Universal Robots URScript: LensSpacer.script

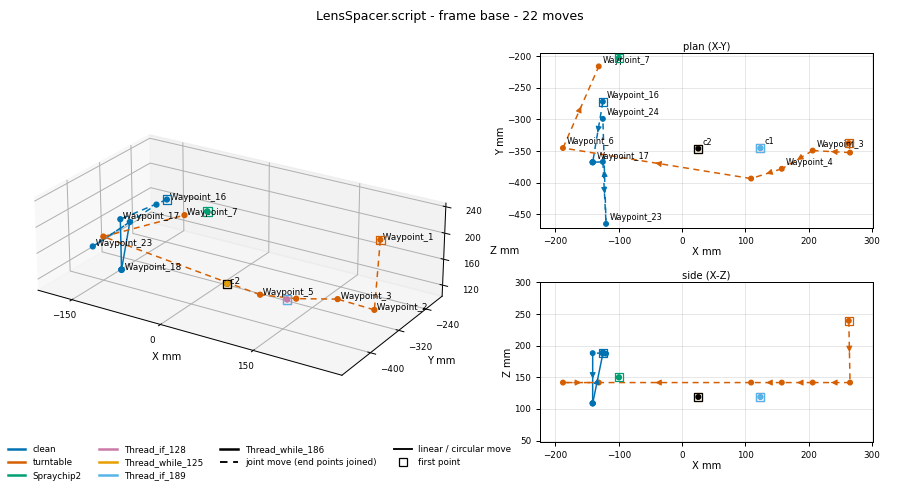
[picture p0: tool path of LensSpacer.script in frame base, 22 of 66 moves have a stored position in this frame; points joined in program order, loops and branches not executed]
def LensSpacer():
  global _hidden_verificationVariable=0
  step_count_fb48d3ff_0c9f_4d99_a765_ea41926c28d5 = 0.0
  thread Step_Counter_Thread_a9617a2c_6c0b_4ca4_aaba_c79477845290():
    while (True):
      step_count_fb48d3ff_0c9f_4d99_a765_ea41926c28d5 = step_count_fb48d3ff_0c9f_4d99_a765_ea41926c28d5 + 1.0
      sync()
    end
  end
  run Step_Counter_Thread_a9617a2c_6c0b_4ca4_aaba_c79477845290()
  set_standard_analog_input_domain(0, 1)
  set_standard_analog_input_domain(1, 1)
  set_tool_analog_input_domain(0, 1)
  set_tool_analog_input_domain(1, 1)
  set_analog_outputdomain(0, 0)
  set_analog_outputdomain(1, 0)
  set_input_actions_to_default()
  set_tool_communication(False, 115200, 0, 1, 1.5, 3.5)
  set_tool_output_mode(0)
  set_tool_digital_output_mode(0, 1)
  set_tool_digital_output_mode(1, 1)
  set_tool_voltage(0)
  set_safety_mode_transition_hardness(1)
  set_gravity([0.0, 0.0, 9.82])
  set_target_payload(0.530000, [0.009000, -0.039000, 0.092000], [0.000534, 0.000534, 0.000534, 0.000000, 0.000000, 0.000000])
  set_tcp(p[0.0,0.0,0.11,0.0,0.0,0.0])
  global Al_plate=p[0.12405209206180495,-0.2666666051843552,0.020008101224669964,-9.276623980477388E-5,1.8107917580596192E-5,3.1233857134705927]
  global Frame2x2=p[0.18266245434305164,-0.34273121659514855,0.026002571110600767,-2.225423529876215E-4,3.0110667546023537E-4,3.1233976058306383]
  global Plane_1=p[0.0,0.0,0.0,0.0,0.0,0.0]
  global URlogoTutorial=p[-0.08178353973148575,-0.3363174165299142,0.04788621506469384,-3.9746155723688456E-5,-3.4682148779121894E-5,-1.5668291789091222]
  global carousel=p[0.13865255139760183,-0.25132593351268107,0.051531504137083003,-4.453572132438073E-5,-1.3071222590669835E-4,-3.1349676625391965]
  global carouselrod=p[0.2020731702281844,-0.34951442511341274,0.1947611446273096,3.139766958234101,-0.10689428010274801,-1.1796370330365635E-5]
  global paper=p[-0.09670794781244417,-0.3283412964648025,0.027665994240809913,-3.2057893450593004E-5,2.867088716161181E-5,-1.6085327915291054]
  global rod=p[0.13368013097420872,-0.41123185103490206,0.09926814901395645,2.2214229924093103,-2.2214158162465862,-2.9165882738638143E-5]
  global timer_1=0
  global c1_p=p[.123835058239, -.345418431995, .118986505182, -3.106795474555, -.465619356567, .000150367177]
  global c1_q=[-0.8607562224017542, -1.7996555767455042, -1.6686586141586304, -1.243450478916504, 1.5722103118896484, 3.55291748046875]
  global c2_p=p[.025685349615, -.346070581208, .119008047533, -3.141142372007, .028389149609, .002727345742]
  global c2_q=[-1.1080010573016565, -1.7158266506590785, -1.7707760334014893, -1.2261001926711579, 1.5707616806030273, 3.621312379837036]
  global Waypoint_16_p=p[-.125097928533, -.271984222044, .188211676824, -3.139810722578, .105446315311, .000070958927]
  global Waypoint_16_q=[-1.5480602423297327, -1.4491210740855713, -1.7099264860153198, -1.552596167927124, 1.5715936422348022, 3.23006010055542]
  global Waypoint_17_p=p[-.141183217597, -.367684006591, .188213447751, 3.139821760490, -.105397104768, -.000067867997]
  global Waypoint_17_q=[-1.597567383443014, -1.8740092716612757, -1.241610050201416, -1.5960084400572718, 1.5719740390777588, 3.1803600788116455]
  global Waypoint_18_p=p[-.141178244459, -.367687282910, .108904454765, 3.139816402425, -.105408093734, -.000060814483]
  global Waypoint_18_q=[-1.5975983778582972, -1.9245020351805628, -1.550661325454712, -1.2364590925029297, 1.5723340511322021, 3.1807193756103516]
  global Waypoint_19_p=p[-.141189357305, -.367687267469, .108915260822, 3.121780755938, .351957921543, -.000099281586]
  global Waypoint_19_q=[-1.5976179281817835, -1.9244748554625453, -1.550661325454712, -1.2364507478526612, 1.572314977645874, 2.889045000076294]
  global Waypoint_20_p=p[-.141176698746, -.367682773595, .108907204798, -3.111042719163, .436975672702, .000063164110]
  global Waypoint_20_q=[-1.5975945631610315, -1.9244939289488734, -1.5506495237350464, -1.2365017098239441, 1.5723340511322021, 3.3926987648010254]
  global Waypoint_21_p=p[-.141174078526, -.367696805030, .108909057026, 3.139786221315, -.105395786134, -.000060564502]
  global Waypoint_21_q=[-1.597586456929342, -1.9245058498778285, -1.5506460666656494, -1.2364399594119568, 1.5723340511322021, 3.1807241439819336]
  global Waypoint_22_p=p[-.125093999497, -.367099400456, .187371407622, 3.139783011421, -.105392168035, -.000053869150]
  global Waypoint_22_q=[-1.5538747946368616, -1.846323629418844, -1.2822730541229248, -1.5829936466612757, 1.5719654560089111, 3.224064588546753]
  global Waypoint_23_p=p[-.120064390322, -.465070651334, .187365924664, 2.700279766902, -.088400420341, .019763045538]
  global Waypoint_23_q=[-1.5412524382220667, -1.9475652180113734, -1.406833291053772, -0.9173591893962403, 1.5603561401367188, 3.2332537174224854]
  global Waypoint_24_p=p[-.125099110421, -.299097154487, .189878767902, 3.139750209928, -.105401717856, -.000111797080]
  global Waypoint_24_q=[-1.550074879323141, -1.5617311683348198, -1.5979981422424316, -1.5518303674510499, 1.5716702938079834, 3.2279696464538574]
  global Waypoint_1_p=p[.263501689877, -.337317763427, .239349489480, 3.139797243720, -.105347053477, -.000037720516]
  global Waypoint_1_q=[-0.5959728399859827, -2.1057659588255824, -0.6533136367797852, -1.9525557957091273, 1.5718059539794922, 4.181682586669922]
  global Waypoint_2_p=p[.265438435610, -.352444474661, .141740907029, 3.139726376264, -.105360108121, -.000022031768]
  global Waypoint_2_q=[-0.6231134573565882, -2.1016999683775843, -1.126999020576477, -1.4828875821879883, 1.5722739696502686, 4.154912948608398]
  global Waypoint_3_p=p[.206441973084, -.349241721273, .141737893294, 3.139734184252, -.105329347268, -.000022485776]
  global Waypoint_3_q=[-0.7073677221881312, -1.9410401783385218, -1.3681066036224365, -1.4024366003325959, 1.5721865892410278, 4.070710182189941]
  global Waypoint_4_p=p[.157616611756, -.378012026932, .141738203587, 3.139764187573, -.105376653239, -.000076760662]
  global Waypoint_4_q=[-0.8494070211993616, -1.9579774341978968, -1.3439116477966309, -1.409730003481247, 1.5722019672393799, 3.928692579269409]
  global Waypoint_5_p=p[.109134761588, -.393436595889, .141742225598, 3.139732501163, -.105376381431, -.000050533951]
  global Waypoint_5_q=[-0.972816292439596, -1.9523960552611292, -1.3519116640090942, -1.4072665137103577, 1.5721949338912964, 3.805286407470703]
  global Waypoint_6_p=p[-.188131250090, -.345166366147, .141750553976, 3.139727051239, -.105353578209, -.000024875816]
  global Waypoint_6_q=[-1.7293437162982386, -1.8864180050291957, -1.4439769983291626, -1.381135032778122, 1.572224736213684, 3.0487747192382812]
  global Waypoint_7_p=p[-.131564048097, -.216205376465, .141741700579, 3.139714533984, -.105382776464, -.000044168049]
  global Waypoint_7_q=[-1.572542969380514, -1.2417927545360108, -2.0833356380462646, -1.3863917154124756, 1.571577787399292, 3.2058310508728027]
  global chipC_p=p[-.099697868296, -.202950013539, .149999031187, 3.139665329235, -.105467028523, -.000070092891]
  global chipC_q=[-1.408487621937887, -1.0837985140136261, -2.130019187927246, -1.497666673069336, 1.571320652961731, 3.369939088821411]
  global timer_1_is_counting=False
  thread Timer_Thread():
    while (True):
      if (timer_1_is_counting):
        timer_1 = timer_1 + get_steptime()
      end
      sync()
    end
  end
  run Timer_Thread()
  def CircleAllangles():
    $ 258 "CircleAllangles" "noBreak"
    $ 259 "p0≔p[c[0]+r,c[1],c[2],c[3],c[4],c[5]-1.5*A]"
    global p0=p[c[0]+r,c[1],c[2],c[3],c[4],c[5]-1.5*A]
    $ 260 "p45≔p[c[0]+0.71*r,c[1]+0.71*r,c[2],c[3]-A/1.1,c[4],c[5]-A/1.1]"
    global p45=p[c[0]+0.71*r,c[1]+0.71*r,c[2],c[3]-A/1.1,c[4],c[5]-A/1.1]
    $ 261 "p90≔p[c[0],c[1]+r,c[2],c[3]-A,c[4],c[5]]"
    global p90=p[c[0],c[1]+r,c[2],c[3]-A,c[4],c[5]]
    $ 262 "p135≔p[c[0]-0.71*r,c[1]+0.71*r,c[2],c[3]-A/1.1,c[4],c[5]+A/1.1]"
    global p135=p[c[0]-0.71*r,c[1]+0.71*r,c[2],c[3]-A/1.1,c[4],c[5]+A/1.1]
    $ 263 "p180≔p[c[0]-r,c[1],c[2],c[3],c[4],c[5]+1.5*A]"
    global p180=p[c[0]-r,c[1],c[2],c[3],c[4],c[5]+1.5*A]
    $ 264 "p225≔p[c[0]-0.71*r,c[1]-0.71*r,c[2],c[3]+A/1.1,c[4],c[5]+A/1.1]"
    global p225=p[c[0]-0.71*r,c[1]-0.71*r,c[2],c[3]+A/1.1,c[4],c[5]+A/1.1]
    $ 265 "p270≔p[c[0],c[1]-r,c[2],c[3]+A,c[4],c[5]]"
    global p270=p[c[0],c[1]-r,c[2],c[3]+A,c[4],c[5]]
    $ 266 "p315≔p[c[0]+0.71*r,c[1]-0.71*r,c[2],c[3]+A/1.1,c[4],c[5]-A/1.1]"
    global p315=p[c[0]+0.71*r,c[1]-0.71*r,c[2],c[3]+A/1.1,c[4],c[5]-A/1.1]
    $ 267 "Set atomization=On"
    set_standard_digital_out(1, True)
    $ 268 "Set triggersolenoid=On"
    set_standard_digital_out(0, True)
    $ 269 "MoveL"
    $ 270 "p0" "breakAfter"
    set_tcp(p[0.0,0.0,0.11,0.0,0.0,0.0])
    movel(p0, a=1.3, v=0.4, r=0.005)
    $ 271 "p45" "breakAfter"
    set_tcp(p[0.0,0.0,0.11,0.0,0.0,0.0])
    movel(p45, a=1.3, v=0.4, r=0.005)
    $ 272 "p90" "breakAfter"
    set_tcp(p[0.0,0.0,0.11,0.0,0.0,0.0])
    movel(p90, a=1.3, v=0.4, r=0.005)
    $ 273 "p135" "breakAfter"
    set_tcp(p[0.0,0.0,0.11,0.0,0.0,0.0])
    movel(p135, a=1.3, v=0.4, r=0.005)
    $ 274 "p180" "breakAfter"
    set_tcp(p[0.0,0.0,0.11,0.0,0.0,0.0])
    movel(p180, a=1.3, v=0.4, r=0.005)
    $ 275 "p225" "breakAfter"
    set_tcp(p[0.0,0.0,0.11,0.0,0.0,0.0])
    movel(p225, a=1.3, v=0.4, r=0.005)
    $ 276 "p270" "breakAfter"
    set_tcp(p[0.0,0.0,0.11,0.0,0.0,0.0])
    movel(p270, a=1.3, v=0.4, r=0.005)
    $ 277 "p315" "breakAfter"
    set_tcp(p[0.0,0.0,0.11,0.0,0.0,0.0])
    movel(p315, a=1.3, v=0.4, r=0.005)
    $ 278 "p0" "breakAfter"
    set_tcp(p[0.0,0.0,0.11,0.0,0.0,0.0])
    movel(p0, a=1.3, v=0.4, r=0.005)
    $ 279 "p45" "breakAfter"
    set_tcp(p[0.0,0.0,0.11,0.0,0.0,0.0])
    movel(p45, a=1.3, v=0.4, r=0.005)
    $ 280 "p90" "breakAfter"
    set_tcp(p[0.0,0.0,0.11,0.0,0.0,0.0])
    movel(p90, a=1.3, v=0.4, r=0.005)
    $ 281 "Set atomization=Off"
    set_standard_digital_out(1, False)
    $ 282 "Set triggersolenoid=Off"
    set_standard_digital_out(0, False)
  end
  def clean():
    $ 283 "clean" "noBreak"
    $ 284 "MoveJ"
    $ 285 "Waypoint_16" "breakAfter"
    movej(get_inverse_kin(Waypoint_16_p, qnear=Waypoint_16_q), a=1.3962634015954636, v=1.0471975511965976)
    $ 286 "Waypoint_17" "breakAfter"
    movej(get_inverse_kin(Waypoint_17_p, qnear=Waypoint_17_q), a=1.3962634015954636, v=1.0471975511965976)
    $ 287 "MoveL"
    $ 288 "Waypoint_18" "breakAfter"
    movel(Waypoint_18_p, a=1.2, v=0.05)
    $ 289 "MoveL"
    $ 290 "Waypoint_19" "breakAfter"
    movel(Waypoint_19_p, a=1.2, v=0.05)
    $ 291 "MoveL"
    $ 292 "Waypoint_20" "breakAfter"
    movel(Waypoint_20_p, a=1.2, v=0.05)
    $ 293 "MoveL"
    $ 294 "Waypoint_21" "breakAfter"
    movel(Waypoint_21_p, a=1.2, v=0.05)
    $ 295 "MoveL"
    $ 296 "Waypoint_22" "breakAfter"
    movel(Waypoint_22_p, a=1.2, v=0.25)
    $ 297 "MoveJ"
    $ 298 "Waypoint_23" "breakAfter"
    movej(get_inverse_kin(Waypoint_23_p, qnear=Waypoint_23_q), a=1.3962634015954636, v=1.0471975511965976)
    $ 299 "Set atomization=On"
    set_standard_digital_out(1, True)
    $ 300 "Set triggersolenoid=On"
    set_standard_digital_out(0, True)
    $ 301 "Wait: 0.2"
    sleep(0.2)
    $ 302 "Set atomization=Off"
    set_standard_digital_out(1, False)
    $ 303 "Set triggersolenoid=Off"
    set_standard_digital_out(0, False)
    $ 304 "MoveJ"
    $ 305 "Waypoint_24" "breakAfter"
    movej(get_inverse_kin(Waypoint_24_p, qnear=Waypoint_24_q), a=1.3962634015954636, v=1.0471975511965976)
  end
  def turntable():
    $ 306 "turntable" "noBreak"
    $ 307 "MoveJ"
    $ 308 "Waypoint_1" "breakAfter"
    set_tcp(p[0.0,0.0,0.11,0.0,0.0,0.0])
    movej(get_inverse_kin(pose_trans(carouselrod, pose_trans(p[-.225374943892, -.334963115589, .194760490875, -3.139766958133, .106894280099, .000011796372], Waypoint_1_p)), qnear=Waypoint_1_q), a=1.3962634015954636, v=0.5235987755982988, r=0.02)
    $ 309 "Waypoint_2" "breakAfter"
    set_tcp(p[0.0,0.0,0.11,0.0,0.0,0.0])
    movej(get_inverse_kin(pose_trans(carouselrod, pose_trans(p[-.225374943892, -.334963115589, .194760490875, -3.139766958133, .106894280099, .000011796372], Waypoint_2_p)), qnear=Waypoint_2_q), a=1.3962634015954636, v=0.5235987755982988, r=0.02)
    $ 310 "Waypoint_3" "breakAfter"
    set_tcp(p[0.0,0.0,0.11,0.0,0.0,0.0])
    movej(get_inverse_kin(pose_trans(carouselrod, pose_trans(p[-.225374943892, -.334963115589, .194760490875, -3.139766958133, .106894280099, .000011796372], Waypoint_3_p)), qnear=Waypoint_3_q), a=1.3962634015954636, v=0.5235987755982988, r=0.02)
    $ 311 "Waypoint_4" "breakAfter"
    set_tcp(p[0.0,0.0,0.11,0.0,0.0,0.0])
    movej(get_inverse_kin(pose_trans(carouselrod, pose_trans(p[-.225374943892, -.334963115589, .194760490875, -3.139766958133, .106894280099, .000011796372], Waypoint_4_p)), qnear=Waypoint_4_q), a=1.3962634015954636, v=0.5235987755982988, r=0.02)
    $ 312 "Waypoint_5" "breakAfter"
    set_tcp(p[0.0,0.0,0.11,0.0,0.0,0.0])
    movej(get_inverse_kin(pose_trans(carouselrod, pose_trans(p[-.225374943892, -.334963115589, .194760490875, -3.139766958133, .106894280099, .000011796372], Waypoint_5_p)), qnear=Waypoint_5_q), a=1.3962634015954636, v=0.5235987755982988, r=0.02)
    $ 313 "MoveJ"
    $ 314 "Waypoint_6" "breakAfter"
    movej(get_inverse_kin(pose_trans(carouselrod, pose_trans(p[-.225374943892, -.334963115589, .194760490875, -3.139766958133, .106894280099, .000011796372], Waypoint_6_p)), qnear=Waypoint_6_q), a=1.3962634015954636, v=0.3141592653589793)
    $ 315 "Wait: 1.0"
    sleep(1.0)
    $ 316 "MoveJ"
    $ 317 "Waypoint_7" "breakAfter"
    movej(get_inverse_kin(pose_trans(carouselrod, pose_trans(p[-.225374943892, -.334963115589, .194760490875, -3.139766958133, .106894280099, .000011796372], Waypoint_7_p)), qnear=Waypoint_7_q), a=1.3962634015954636, v=1.0471975511965976, r=0.02)
  end
  def Spraychip2():
    $ 318 "Spraychip2" "noBreak"
    $ 319 "MoveJ"
    $ 320 "chipC" "breakAfter"
    movej(get_inverse_kin(chipC_p, qnear=chipC_q), a=1.3962634015954636, v=1.0471975511965976)
    $ 321 "c≔chipC"
    global c=chipC_p
    $ 322 "rc≔27/1000"
    global rc=27/1000
    $ 323 "p0≔p[c[0]+rc,c[1],c[2],c[3],c[4],c[5]-1.5*0]"
    global p0=p[c[0]+rc,c[1],c[2],c[3],c[4],c[5]-1.5*0]
    $ 324 "p45≔p[c[0]+0.71*rc,c[1]+0.71*rc,c[2],c[3]-0/1.1,c[4],c[5]-0/1.1]"
    global p45=p[c[0]+0.71*rc,c[1]+0.71*rc,c[2],c[3]-0/1.1,c[4],c[5]-0/1.1]
    $ 325 "p90≔p[c[0],c[1]+rc,c[2],c[3]-0,c[4],c[5]]"
    global p90=p[c[0],c[1]+rc,c[2],c[3]-0,c[4],c[5]]
    $ 326 "p135≔p[c[0]-0.71*rc,c[1]+0.71*rc,c[2],c[3]-0/1.1,c[4],c[5]+0/1.1]"
    global p135=p[c[0]-0.71*rc,c[1]+0.71*rc,c[2],c[3]-0/1.1,c[4],c[5]+0/1.1]
    $ 327 "p180≔p[c[0]-rc,c[1],c[2],c[3],c[4],c[5]+1.5*0]"
    global p180=p[c[0]-rc,c[1],c[2],c[3],c[4],c[5]+1.5*0]
    $ 328 "p225≔p[c[0]-0.71*rc,c[1]-0.71*rc,c[2],c[3]+0/1.1,c[4],c[5]+0/1.1]"
    global p225=p[c[0]-0.71*rc,c[1]-0.71*rc,c[2],c[3]+0/1.1,c[4],c[5]+0/1.1]
    $ 329 "p270≔p[c[0],c[1]-rc,c[2],c[3]+0,c[4],c[5]]"
    global p270=p[c[0],c[1]-rc,c[2],c[3]+0,c[4],c[5]]
    $ 330 "p315≔p[c[0]+0.71*rc,c[1]-0.71*rc,c[2],c[3]+0/1.1,c[4],c[5]-0/1.1]"
    global p315=p[c[0]+0.71*rc,c[1]-0.71*rc,c[2],c[3]+0/1.1,c[4],c[5]-0/1.1]
    $ 331 "Set atomization=On"
    set_standard_digital_out(1, True)
    $ 332 "Set triggersolenoid=On"
    set_standard_digital_out(0, True)
    $ 333 "MoveL"
    $ 334 "p0" "breakAfter"
    set_tcp(p[0.0,0.0,0.11,0.0,0.0,0.0])
    movel(p0, a=1.3, v=0.085, r=0.01)
    $ 335 "p45" "breakAfter"
    set_tcp(p[0.0,0.0,0.11,0.0,0.0,0.0])
    movel(p45, a=1.3, v=0.085, r=0.01)
    $ 336 "p90" "breakAfter"
    set_tcp(p[0.0,0.0,0.11,0.0,0.0,0.0])
    movel(p90, a=1.3, v=0.085, r=0.01)
    $ 337 "p135" "breakAfter"
    set_tcp(p[0.0,0.0,0.11,0.0,0.0,0.0])
    movel(p135, a=1.3, v=0.085, r=0.01)
    $ 338 "p180" "breakAfter"
    set_tcp(p[0.0,0.0,0.11,0.0,0.0,0.0])
    movel(p180, a=1.3, v=0.085, r=0.01)
    $ 339 "Set triggersolenoid=Off"
    set_standard_digital_out(0, False)
    $ 340 "Wait: 0.1"
    sleep(0.1)
    $ 341 "Set triggersolenoid=On"
    set_standard_digital_out(0, True)
    $ 342 "p225" "breakAfter"
    set_tcp(p[0.0,0.0,0.11,0.0,0.0,0.0])
    movel(p225, a=1.3, v=0.085, r=0.01)
    $ 343 "p270" "breakAfter"
    set_tcp(p[0.0,0.0,0.11,0.0,0.0,0.0])
    movel(p270, a=1.3, v=0.085, r=0.01)
    $ 344 "p315" "breakAfter"
    set_tcp(p[0.0,0.0,0.11,0.0,0.0,0.0])
    movel(p315, a=1.3, v=0.085, r=0.01)
    $ 345 "p0" "breakAfter"
    set_tcp(p[0.0,0.0,0.11,0.0,0.0,0.0])
    movel(p0, a=1.3, v=0.085, r=0.01)
    $ 346 "p45" "breakAfter"
    set_tcp(p[0.0,0.0,0.11,0.0,0.0,0.0])
    movel(p45, a=1.3, v=0.085, r=0.01)
    $ 347 "Set triggersolenoid=Off"
    set_standard_digital_out(0, False)
    $ 348 "Wait: 0.1"
    sleep(0.1)
    $ 349 "Set triggersolenoid=On"
    set_standard_digital_out(0, True)
    $ 350 "p90" "breakAfter"
    set_tcp(p[0.0,0.0,0.11,0.0,0.0,0.0])
    movel(p90, a=1.3, v=0.085, r=0.01)
    $ 351 "p135" "breakAfter"
    set_tcp(p[0.0,0.0,0.11,0.0,0.0,0.0])
    movel(p135, a=1.3, v=0.085, r=0.01)
    $ 352 "p180" "breakAfter"
    set_tcp(p[0.0,0.0,0.11,0.0,0.0,0.0])
    movel(p180, a=1.3, v=0.085, r=0.01)
    $ 353 "p225" "breakAfter"
    set_tcp(p[0.0,0.0,0.11,0.0,0.0,0.0])
    movel(p225, a=1.3, v=0.085, r=0.01)
    $ 354 "p270" "breakAfter"
    set_tcp(p[0.0,0.0,0.11,0.0,0.0,0.0])
    movel(p270, a=1.3, v=0.085, r=0.01)
    $ 355 "p315" "breakAfter"
    set_tcp(p[0.0,0.0,0.11,0.0,0.0,0.0])
    movel(p315, a=1.3, v=0.085, r=0.01)
    $ 356 "p0" "breakAfter"
    set_tcp(p[0.0,0.0,0.11,0.0,0.0,0.0])
    movel(p0, a=1.3, v=0.085, r=0.01)
    $ 357 "MoveJ"
    $ 358 "chipC" "breakAfter"
    movej(get_inverse_kin(chipC_p, qnear=chipC_q), a=1.3962634015954636, v=1.0471975511965976)
    $ 359 "Wait: 0.2"
    sleep(0.2)
    $ 360 "Set atomization=Off"
    set_standard_digital_out(1, False)
    $ 361 "Set triggersolenoid=Off"
    set_standard_digital_out(0, False)
  end
  while (True):
    $ 2 "Robot Program"
    $ 3 "'Program to be used for part #124517-009 lens spacer'"
    # 'Program to be used for part #124517-009 lens spacer'
    $ 4 "'Program rev A: 8/21/24 equalized spray center heights to -281mm in view perspective (c1 was -257mm previously)'"
    # 'Program rev A: 8/21/24 equalized spray center heights to -281mm in view perspective (c1 was -257mm previously)'
    $ 5 "'Program rev B: 8/28/24 added compatibility with stacked masks and adjusted chip spray height to better respresent parts'"
    # 'Program rev B: 8/28/24 added compatibility with stacked masks and adjusted chip spray height to better respresent parts'
    $ 6 "timer_1: Start"
    timer_1_is_counting = True
    $ 7 "r≔1/1000"
    global r=1/1000
    $ 8 "A≔8*3.1416/180"
    global A=8*3.1416/180
    $ 11 "sidenum≔2"
    global sidenum=2
    $ 13 "coatnum≔2"
    global coatnum=2
    $ 15 "partnum≔2"
    global partnum=2
    $ 16 "stack≔'Are masks stacked in 2s?'"
    global stack=request_boolean_from_primary_client("Are masks stacked in 2s?")
    $ 17 "Loop_1≔1"
    global Loop_1=1
    $ 121 "If partnum≤sidenum"
    global thread_flag_121=0
    thread Thread_if_121():
      $ 122 "Loop (coatnum)>0"
      thread Thread_while_122():
        while (True):
          $ 123 "partleft≔partnum"
          global partleft=partnum
          $ 124 "loopnum≔1"
          global loopnum=1
          $ 125 "Loop partleft>0"
          thread Thread_while_125():
            while (True):
              $ 126 "Call clean"
              clean()
              $ 127 "Call Spraychip2"
              Spraychip2()
              $ 128 "If loopnum≟1 or loopnum≟3 or loopnum≟5 or loopnum≟7 or loopnum≟9 or loopnum≟11"
              global thread_flag_128=0
              thread Thread_if_128():
                $ 129 "MoveJ"
                $ 130 "c1" "breakAfter"
                movej(get_inverse_kin(c1_p, qnear=c1_q), a=1.3962634015954636, v=1.0471975511965976)
                $ 131 "c≔c1"
                global c=c1_p
                $ 132 "If stack≟ True "
                if (stack ==   True  ):
                  $ 133 "c≔p[c[0],c[1],c[2]+10/1000,c[3],c[4],c[5]]"
                  global c=p[c[0],c[1],c[2]+10/1000,c[3],c[4],c[5]]
                  $ 134 "MoveL"
                  $ 135 "c" "breakAfter"
                  movel(c, a=1.2, v=0.25)
                end
                $ 136 "Call CircleAllangles"
                CircleAllangles()
                $ 137 "x2≔p[c[0]-0.037,c[1],c[2],c[3],c[4],c[5]]"
                global x2=p[c[0]-0.037,c[1],c[2],c[3],c[4],c[5]]
                $ 138 "x3≔p[c[0]-0.037,c[1]+0.037,c[2],c[3],c[4],c[5]]"
                global x3=p[c[0]-0.037,c[1]+0.037,c[2],c[3],c[4],c[5]]
                $ 139 "x4≔p[c[0],c[1]+0.037,c[2],c[3],c[4],c[5]]"
                global x4=p[c[0],c[1]+0.037,c[2],c[3],c[4],c[5]]
                $ 140 "MoveJ"
                $ 141 "x2" "breakAfter"
                movej(x2, a=1.3962634015954636, v=1.0471975511965976)
                $ 142 "c≔x2"
                global c=x2
                $ 143 "Call CircleAllangles"
                CircleAllangles()
                $ 144 "MoveJ"
                $ 145 "x3" "breakAfter"
                movej(x3, a=1.3962634015954636, v=1.0471975511965976)
                $ 146 "c≔x3"
                global c=x3
                $ 147 "Call CircleAllangles"
                CircleAllangles()
                $ 148 "MoveJ"
                $ 149 "x4" "breakAfter"
                movej(x4, a=1.3962634015954636, v=1.0471975511965976)
                $ 150 "c≔x4"
                global c=x4
                $ 151 "Call CircleAllangles"
                CircleAllangles()
                thread_flag_128 = 1
              end
              if (loopnum == 1  or  loopnum == 3  or  loopnum == 5  or  loopnum == 7  or  loopnum == 9  or  loopnum == 11):
                global thread_handler_128=run Thread_if_128()
                while (thread_flag_128 == 0):
                  if not(loopnum == 1  or  loopnum == 3  or  loopnum == 5  or  loopnum == 7  or  loopnum == 9  or  loopnum == 11):
                    kill thread_handler_128
                    thread_flag_128 = 2
                  else:
                    sync()
                  end
                end
              else:
                thread_flag_128 = 2
              end
              if (thread_flag_128 == 2):
                $ 152 "Else" "noBreak"
                $ 153 "MoveJ"
                $ 154 "c2" "breakAfter"
                movej(get_inverse_kin(c2_p, qnear=c2_q), a=1.3962634015954636, v=1.0471975511965976)
                $ 155 "c≔c2"
                global c=c2_p
                $ 156 "If stack≟ True "
                if (stack ==   True  ):
                  $ 157 "c≔p[c[0],c[1],c[2]+10/1000,c[3],c[4],c[5]]"
                  global c=p[c[0],c[1],c[2]+10/1000,c[3],c[4],c[5]]
                  $ 158 "MoveL"
                  $ 159 "c" "breakAfter"
                  movel(c, a=1.2, v=0.25)
                end
                $ 160 "Call CircleAllangles"
                CircleAllangles()
                $ 161 "x2≔p[c[0]-0.037,c[1],c[2],c[3],c[4],c[5]]"
                global x2=p[c[0]-0.037,c[1],c[2],c[3],c[4],c[5]]
                $ 162 "x3≔p[c[0]-0.037,c[1]+0.037,c[2],c[3],c[4],c[5]]"
                global x3=p[c[0]-0.037,c[1]+0.037,c[2],c[3],c[4],c[5]]
                $ 163 "x4≔p[c[0],c[1]+0.037,c[2],c[3],c[4],c[5]]"
                global x4=p[c[0],c[1]+0.037,c[2],c[3],c[4],c[5]]
                $ 164 "MoveJ"
                $ 165 "x2" "breakAfter"
                movej(x2, a=1.3962634015954636, v=1.0471975511965976)
                $ 166 "c≔x2"
                global c=x2
                $ 167 "Call CircleAllangles"
                CircleAllangles()
                $ 168 "MoveJ"
                $ 169 "x3" "breakAfter"
                movej(x3, a=1.3962634015954636, v=1.0471975511965976)
                $ 170 "c≔x3"
                global c=x3
                $ 171 "Call CircleAllangles"
                CircleAllangles()
                $ 172 "MoveJ"
                $ 173 "x4" "breakAfter"
                movej(x4, a=1.3962634015954636, v=1.0471975511965976)
                $ 174 "c≔x4"
                global c=x4
                $ 175 "Call CircleAllangles"
                CircleAllangles()
              end
              $ 176 "loopnum≔loopnum+1"
              global loopnum=loopnum+1
              $ 177 "partleft≔partleft-1"
              global partleft=partleft-1
            end
          end
          if (partleft>0):
            global thread_handler_125=run Thread_while_125()
            while (partleft>0):
              sync()
            end
            kill thread_handler_125
          end
          $ 178 "i≔0"
          global i=0
          $ 179 "coatnum≔coatnum-1"
          global coatnum=coatnum-1
        end
      end
      if ((coatnum)>0):
        global thread_handler_122=run Thread_while_122()
        while ((coatnum)>0):
          sync()
        end
        kill thread_handler_122
      end
      $ 180 "Halt"
      halt
      thread_flag_121 = 1
    end
    if (partnum <= sidenum):
      global thread_handler_121=run Thread_if_121()
      while (thread_flag_121 == 0):
        if not(partnum <= sidenum):
          kill thread_handler_121
          thread_flag_121 = 2
        else:
          sync()
        end
      end
    else:
      thread_flag_121 = 2
    end
    if (thread_flag_121 == 2):
      $ 181 "Else" "noBreak"
      $ 182 "Loop (coatnum)>0"
      thread Thread_while_182():
        while (True):
          $ 183 "partleft≔partnum"
          global partleft=partnum
          $ 184 "loopnum≔1"
          global loopnum=1
          $ 185 "turnnum≔0"
          global turnnum=0
          $ 186 "Loop partleft>0"
          thread Thread_while_186():
            while (True):
              $ 187 "Call clean"
              clean()
              $ 188 "Call Spraychip2"
              Spraychip2()
              $ 189 "If loopnum≟1 or loopnum≟3 or loopnum≟5 or loopnum≟7 or loopnum≟9 or loopnum≟11"
              global thread_flag_189=0
              thread Thread_if_189():
                $ 190 "MoveJ"
                $ 191 "c1" "breakAfter"
                movej(get_inverse_kin(c1_p, qnear=c1_q), a=1.3962634015954636, v=1.0471975511965976)
                $ 192 "c≔c1"
                global c=c1_p
                $ 193 "If stack≟ True "
                if (stack ==   True  ):
                  $ 194 "c≔p[c[0],c[1],c[2]+10/1000,c[3],c[4],c[5]]"
                  global c=p[c[0],c[1],c[2]+10/1000,c[3],c[4],c[5]]
                  $ 195 "MoveL"
                  $ 196 "c" "breakAfter"
                  movel(c, a=1.2, v=0.25)
                end
                $ 197 "Call CircleAllangles"
                CircleAllangles()
                $ 198 "x2≔p[c[0]-0.037,c[1],c[2],c[3],c[4],c[5]]"
                global x2=p[c[0]-0.037,c[1],c[2],c[3],c[4],c[5]]
                $ 199 "x3≔p[c[0]-0.037,c[1]+0.037,c[2],c[3],c[4],c[5]]"
                global x3=p[c[0]-0.037,c[1]+0.037,c[2],c[3],c[4],c[5]]
                $ 200 "x4≔p[c[0],c[1]+0.037,c[2],c[3],c[4],c[5]]"
                global x4=p[c[0],c[1]+0.037,c[2],c[3],c[4],c[5]]
                $ 201 "MoveJ"
                $ 202 "x2" "breakAfter"
                movej(x2, a=1.3962634015954636, v=1.0471975511965976)
                $ 203 "c≔x2"
                global c=x2
                $ 204 "Call CircleAllangles"
                CircleAllangles()
                $ 205 "MoveJ"
                $ 206 "x3" "breakAfter"
                movej(x3, a=1.3962634015954636, v=1.0471975511965976)
                $ 207 "c≔x3"
                global c=x3
                $ 208 "Call CircleAllangles"
                CircleAllangles()
                $ 209 "MoveJ"
                $ 210 "x4" "breakAfter"
                movej(x4, a=1.3962634015954636, v=1.0471975511965976)
                $ 211 "c≔x4"
                global c=x4
                $ 212 "Call CircleAllangles"
                CircleAllangles()
                thread_flag_189 = 1
              end
              if (loopnum == 1  or  loopnum == 3  or  loopnum == 5  or  loopnum == 7  or  loopnum == 9  or  loopnum == 11):
                global thread_handler_189=run Thread_if_189()
                while (thread_flag_189 == 0):
                  if not(loopnum == 1  or  loopnum == 3  or  loopnum == 5  or  loopnum == 7  or  loopnum == 9  or  loopnum == 11):
                    kill thread_handler_189
                    thread_flag_189 = 2
                  else:
                    sync()
                  end
                end
              else:
                thread_flag_189 = 2
              end
              if (thread_flag_189 == 2):
                $ 213 "Else" "noBreak"
                $ 214 "MoveJ"
                $ 215 "c2" "breakAfter"
                movej(get_inverse_kin(c2_p, qnear=c2_q), a=1.3962634015954636, v=1.0471975511965976)
                $ 216 "c≔c2"
                global c=c2_p
                $ 217 "If stack≟ True "
                if (stack ==   True  ):
                  $ 218 "c≔p[c[0],c[1],c[2]+10/1000,c[3],c[4],c[5]]"
                  global c=p[c[0],c[1],c[2]+10/1000,c[3],c[4],c[5]]
                  $ 219 "MoveL"
                  $ 220 "c" "breakAfter"
                  movel(c, a=1.2, v=0.25)
                end
                $ 221 "Call CircleAllangles"
                CircleAllangles()
                $ 222 "x2≔p[c[0]-0.037,c[1],c[2],c[3],c[4],c[5]]"
                global x2=p[c[0]-0.037,c[1],c[2],c[3],c[4],c[5]]
                $ 223 "x3≔p[c[0]-0.037,c[1]+0.037,c[2],c[3],c[4],c[5]]"
                global x3=p[c[0]-0.037,c[1]+0.037,c[2],c[3],c[4],c[5]]
                $ 224 "x4≔p[c[0],c[1]+0.037,c[2],c[3],c[4],c[5]]"
                global x4=p[c[0],c[1]+0.037,c[2],c[3],c[4],c[5]]
                $ 225 "MoveJ"
                $ 226 "x2" "breakAfter"
                movej(x2, a=1.3962634015954636, v=1.0471975511965976)
                $ 227 "c≔x2"
                global c=x2
                $ 228 "Call CircleAllangles"
                CircleAllangles()
                $ 229 "MoveJ"
                $ 230 "x3" "breakAfter"
                movej(x3, a=1.3962634015954636, v=1.0471975511965976)
                $ 231 "c≔x3"
                global c=x3
                $ 232 "Call CircleAllangles"
                CircleAllangles()
                $ 233 "MoveJ"
                $ 234 "x4" "breakAfter"
                movej(x4, a=1.3962634015954636, v=1.0471975511965976)
                $ 235 "c≔x4"
                global c=x4
                $ 236 "Call CircleAllangles"
                CircleAllangles()
              end
              $ 237 "loopnum≔loopnum+1"
              global loopnum=loopnum+1
              $ 238 "partleft≔partleft-1"
              global partleft=partleft-1
            end
          end
          if (partleft>0):
            global thread_handler_186=run Thread_while_186()
            while (partleft>0):
              sync()
            end
            kill thread_handler_186
          end
          $ 239 "i≔0"
          global i=0
          $ 240 "Loop (6-turnnum)>0"
          thread Thread_while_240():
            while (True):
              $ 241 "Call turntable"
              turntable()
              $ 242 "turnnum≔turnnum+1"
              global turnnum=turnnum+1
            end
          end
          if ((6-turnnum)>0):
            global thread_handler_240=run Thread_while_240()
            while ((6-turnnum)>0):
              sync()
            end
            kill thread_handler_240
          end
          $ 243 "coatnum≔coatnum-1"
          global coatnum=coatnum-1
        end
      end
      if ((coatnum)>0):
        global thread_handler_182=run Thread_while_182()
        while ((coatnum)>0):
          sync()
        end
        kill thread_handler_182
      end
      $ 244 "Halt"
      halt
    end
  end
end
